FUNCTION FC_UpdatePieceCount
VAR_INPUT
	aByte			: stByteAsBit;
	In				: POINTER TO UDINT;
END_VAR

IF FC_ProductStatusNopresence(aByte) = eProductStatus.Completed THEN
	In[eHeaderPieces.Ok] := In[eHeaderPieces.Ok] + 1;
END_IF
IF FC_ProductStatusNopresence(aByte) = eProductStatus.Scraped THEN
	In[eHeaderPieces.Ko] := In[eHeaderPieces.Ko] + 1;
END_IF

END_FUNCTION

(* stored: Version 1.1.0.1, ProductVersion 3.1.4024.15
   POU FC_UpdatePieceCount: Id {3a9d3d10-a702-467c-a024-04e10e9d4318}, SpecialFunc None *)
